KUKA KRL program: f_fraes1.src, f_fraes1.dat

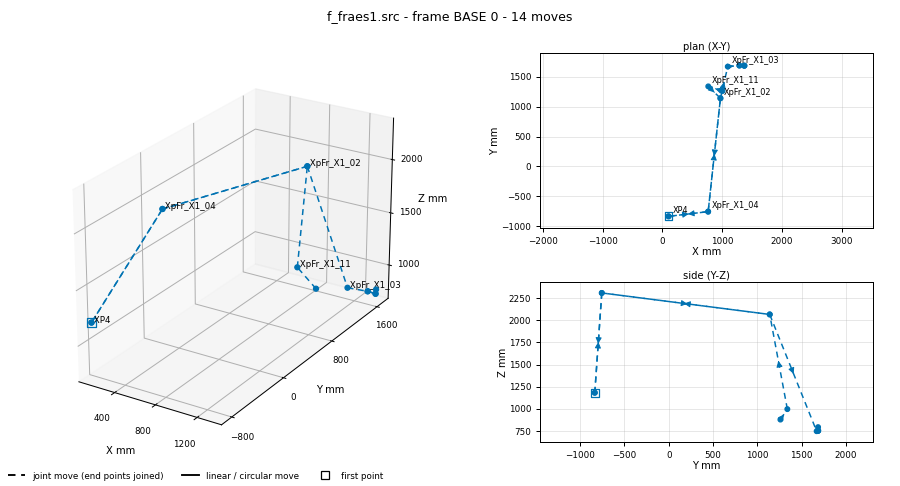
[picture p0: tool path of f_fraes1.src in frame BASE 0, 14 of 15 moves have a stored position in this frame; points joined in program order, loops and branches not executed]
--- f_fraes1.src ---
&ACCESS RVO3
&REL 7
&COMMENT INI Dress X1
&PARAM DISKPATH = KRC:\R1\Program
&PARAM TEMPLATE = C:\KRC\Roboter\Template\vorgabe
&PARAM EDITMASK = *
DEF f_fraes1( )
;FOLD INI
  ;FOLD BASISTECH INI
    GLOBAL INTERRUPT DECL 3 WHEN $STOPMESS==TRUE DO IR_STOPM ( )
    INTERRUPT ON 3
    BAS (#INITMOV,0 )
  ;ENDFOLD (BASISTECH INI)
;FOLD SPOTTECH INI
USERSPOT(#INIT)
;ENDFOLD (SPOTTECH INI)
;FOLD GRIPPERTECH INI
USER_GRP(0,DUMMY,DUMMY,GDEFAULT)
;ENDFOLD (GRIPPERTECH INI)
  ;FOLD USER INI
    ;Make your modifications here

  ;ENDFOLD (USER INI)
;ENDFOLD (INI)

; Caracterização dos meios de produção:
; Versão Atual:
; 08/06/2013 12:00 Name: P13.050-R1 CHANGES: Fresa
; Gun X1 (F2 6640 0018 985)

chk_w1_wechs_ok() ; check X1

;FOLD PTP P4 Vel=100 % PDAT11 Tool[1]:GUN X1 Base[0];%{PE}%R 8.2.20,%MKUKATPBASIS,%CMOVE,%VPTP,%P 1:PTP, 2:P4, 3:, 5:100, 7:PDAT11
$BWDSTART=FALSE
PDAT_ACT=PPDAT11
FDAT_ACT=FP4
BAS(#PTP_PARAMS,100)
PTP XP4
;ENDFOLD

;FOLD PTP pFr_X1_04 CONT Vel=100 % PDAT13 Tool[1]:GUN X1 Base[0];%{PE}%R 8.2.20,%MKUKATPBASIS,%CMOVE,%VPTP,%P 1:PTP, 2:pFr_X1_04, 3:C_DIS, 5:100, 7:PDAT13
$BWDSTART=FALSE
PDAT_ACT=PPDAT13
FDAT_ACT=FpFr_X1_04
BAS(#PTP_PARAMS,100)
PTP XpFr_X1_04 C_DIS
;ENDFOLD
;FOLD PTP pFr_X1_02 CONT Vel=100 % PDAT1 Tool[1]:GUN X1 Base[0];%{PE}%R 8.2.20,%MKUKATPBASIS,%CMOVE,%VPTP,%P 1:PTP, 2:pFr_X1_02, 3:C_DIS, 5:100, 7:PDAT1
$BWDSTART=FALSE
PDAT_ACT=PPDAT1
FDAT_ACT=FpFr_X1_02
BAS(#PTP_PARAMS,100)
PTP XpFr_X1_02 C_DIS
;ENDFOLD
;FOLD PTP pFr_X1_03 CONT Vel=100 % PDAT2 Tool[1]:GUN X1 Base[0];%{PE}%R 8.2.20,%MKUKATPBASIS,%CMOVE,%VPTP,%P 1:PTP, 2:pFr_X1_03, 3:C_DIS, 5:100, 7:PDAT2
$BWDSTART=FALSE
PDAT_ACT=PPDAT2
FDAT_ACT=FpFr_X1_03
BAS(#PTP_PARAMS,100)
PTP XpFr_X1_03 C_DIS
;ENDFOLD
;FOLD PTP pFr_X1_05 CONT Vel=100 % PDAT3 Tool[1]:GUN X1 Base[0];%{PE}%R 8.2.20,%MKUKATPBASIS,%CMOVE,%VPTP,%P 1:PTP, 2:pFr_X1_05, 3:C_DIS, 5:100, 7:PDAT3
$BWDSTART=FALSE
PDAT_ACT=PPDAT3
FDAT_ACT=FpFr_X1_05
BAS(#PTP_PARAMS,100)
PTP XpFr_X1_05 C_DIS
;ENDFOLD
;FOLD LIN pFr_X1_06 Vel=0.25 m/s CPDAT0 Tool[1]:GUN X1 Base[0];%{PE}%R 8.2.20,%MKUKATPBASIS,%CMOVE,%VLIN,%P 1:LIN, 2:pFr_X1_06, 3:, 5:0.25, 7:CPDAT0
$BWDSTART=FALSE
LDAT_ACT=LCPDAT0
FDAT_ACT=FpFr_X1_06
BAS(#CP_PARAMS,0.25)
LIN XpFr_X1_06
;ENDFOLD

;FOLD ; PONTO DE FRESAGEM;%{PE}%R 8.2.20,%MKUKATPBASIS,%CCOMMENT,%VNORMAL,%P 2:PONTO  DE  FRESAGEM
;ENDFOLD
;FOLD TIP.LIN_ Dress5, Spot Gun 4 , RETR open , Tool[1], Base[0], EXT.TCP=FALSE;%{PE}%MKUKATPUSER
FDAT_ACT=FDress5
BAS(#FRAMES)
LIN  XDress5
S_ACT.GUN=4
S_ACT.RETR=#opn
S_READY=FALSE
USERSPOT (#DRESS,S_ACT )
WAIT FOR  S_READY
;ENDFOLD

;FOLD LIN pFr_X1_08 CONT Vel=0.2 m/s CPDAT2 Tool[1]:GUN X1 Base[0];%{PE}%R 8.2.20,%MKUKATPBASIS,%CMOVE,%VLIN,%P 1:LIN, 2:pFr_X1_08, 3:C_DIS C_DIS, 5:0.2, 7:CPDAT2
$BWDSTART=FALSE
LDAT_ACT=LCPDAT2
FDAT_ACT=FpFr_X1_08
BAS(#CP_PARAMS,0.2)
LIN XpFr_X1_08 C_DIS C_DIS
;ENDFOLD
;FOLD LIN pFr_X1_09 CONT Vel=0.35 m/s CPDAT3 Tool[1]:GUN X1 Base[0];%{PE}%R 8.2.20,%MKUKATPBASIS,%CMOVE,%VLIN,%P 1:LIN, 2:pFr_X1_09, 3:C_DIS C_DIS, 5:0.35, 7:CPDAT3
$BWDSTART=FALSE
LDAT_ACT=LCPDAT3
FDAT_ACT=FpFr_X1_09
BAS(#CP_PARAMS,0.35)
LIN XpFr_X1_09 C_DIS C_DIS
;ENDFOLD
;FOLD PTP P3 PDAT10 SPOT Gun=4 RETR OPN PgNo1=254 ACTIVE=1 Tool[1]:GUN X1 Base[1]:Actros;%{PE}%R 8.2.2,%MKUKATPSPOT,%CSPOT,%VPTP,%P 1:PTP, 2:P3, 3:, 5:100, 7:PDAT10, 10:4, 12:#FIRST, 14:#OPN, 16:254, 18:1, 20:0, 22:0, 24:1, 25:NORMAL
$BWDSTART=FALSE
PDAT_ACT=PPDAT10
FDAT_ACT=FP3
BAS(#PTP_PARAMS,PPDAT10.VEL)
S_ACT.GUN=4
S_ACT.PAIR=SDEFAULT.PAIR
S_ACT.RETR=#OPN
S_ACT.CLO_TM=1
S_ACT.PGNO1=254
S_ACT.PGNO2=SDEFAULT.PGNO2
S_ACT.PRESS1=SDEFAULT.PRESS1
S_ACT.PRESS2=SDEFAULT.PRESS2
S_READY=FALSE
PTP XP3
USERSPOT(#SPOT, S_ACT)
WAIT FOR S_READY
;ENDFOLD
;FOLD PTP pFr_X1_10 CONT Vel=100 % PDAT4 Tool[1]:GUN X1 Base[0];%{PE}%R 8.2.20,%MKUKATPBASIS,%CMOVE,%VPTP,%P 1:PTP, 2:pFr_X1_10, 3:C_DIS, 5:100, 7:PDAT4
$BWDSTART=FALSE
PDAT_ACT=PPDAT4
FDAT_ACT=FpFr_X1_10
BAS(#PTP_PARAMS,100)
PTP XpFr_X1_10 C_DIS
;ENDFOLD
;FOLD PTP pFr_X1_11 CONT Vel=100 % PDAT5 Tool[1]:GUN X1 Base[0];%{PE}%R 8.2.20,%MKUKATPBASIS,%CMOVE,%VPTP,%P 1:PTP, 2:pFr_X1_11, 3:C_DIS, 5:100, 7:PDAT5
$BWDSTART=FALSE
PDAT_ACT=PPDAT5
FDAT_ACT=FpFr_X1_11
BAS(#PTP_PARAMS,100)
PTP XpFr_X1_11 C_DIS
;ENDFOLD
;FOLD PTP pFr_X1_12 CONT Vel=100 % PDAT6 Tool[1]:GUN X1 Base[0];%{PE}%R 8.2.20,%MKUKATPBASIS,%CMOVE,%VPTP,%P 1:PTP, 2:pFr_X1_12, 3:C_DIS, 5:100, 7:PDAT6
$BWDSTART=FALSE
PDAT_ACT=PPDAT6
FDAT_ACT=FpFr_X1_12
BAS(#PTP_PARAMS,100)
PTP XpFr_X1_12 C_DIS
;ENDFOLD
;FOLD PTP pFr_X1_07 CONT Vel=100 % PDAT14 Tool[1]:GUN X1 Base[0];%{PE}%R 8.2.20,%MKUKATPBASIS,%CMOVE,%VPTP,%P 1:PTP, 2:pFr_X1_07, 3:C_DIS, 5:100, 7:PDAT14
$BWDSTART=FALSE
PDAT_ACT=PPDAT14
FDAT_ACT=FpFr_X1_07
BAS(#PTP_PARAMS,100)
PTP XpFr_X1_07 C_DIS
;ENDFOLD

;FOLD PTP P5 Vel=100 % PDAT12 Tool[1]:GUN X1 Base[0];%{PE}%R 8.2.20,%MKUKATPBASIS,%CMOVE,%VPTP,%P 1:PTP, 2:P5, 3:, 5:100, 7:PDAT12
$BWDSTART=FALSE
PDAT_ACT=PPDAT12
FDAT_ACT=FP5
BAS(#PTP_PARAMS,100)
PTP XP5
;ENDFOLD

END

--- f_fraes1.dat ---
&ACCESS RVO3
&REL 7
&COMMENT INI Dress X1
&PARAM DISKPATH = KRC:\R1\Program
&PARAM TEMPLATE = C:\KRC\Roboter\Template\vorgabe
&PARAM EDITMASK = *
DEFDAT  f_fraes1
;FOLD EXTERNAL DECLARATIONS;%{PE}%MKUKATPBASIS,%CEXT,%VCOMMON,%P
;FOLD GRIPPERTECH EXT
EXT  H50 (INT  :IN,INT  :IN,INT  :IN,GRP_TYP  :IN )
;ENDFOLD (GRIPPERTECH EXT)
;FOLD SPOTTECH EXT
EXT  USERSPOT (S_COMMAND  :IN,SPOT_TYPE  :IN )
;ENDFOLD (SPOTTECH EXT)
;FOLD BASISTECH EXT;%{PE}%MKUKATPBASIS,%CEXT,%VEXT,%P
EXT  BAS (BAS_COMMAND  :IN,REAL  :IN )
DECL INT SUCCESS
;ENDFOLD (BASISTECH EXT)
;FOLD USER EXT;%{E}%MKUKATPUSER,%CEXT,%VEXT,%P
;Make your modifications here

;ENDFOLD (USER EXT)
;ENDFOLD (EXTERNAL DECLARATIONS)
DECL BASIS_SUGG_T LAST_BASIS={POINT1[] "P5                      ",POINT2[] "P5                      ",CP_PARAMS[] "CPDAT3                  ",PTP_PARAMS[] "PDAT14                  ",CONT[] "                        ",CP_VEL[] "0.35                    ",PTP_VEL[] "100                     ",SYNC_PARAMS[] "SYNCDAT                 ",SPL_NAME[] "S0                      "}
DECL PDAT PPDAT1={VEL 100.0,ACC 100.0,APO_DIST 100.0,APO_MODE #CDIS}
DECL E6POS XpFr_X1_02={X 969.039673,Y 1139.73096,Z 2066.15308,A 44.3954697,B 54.7452507,C 92.8609467,S 2,T 3,E1 199.989594,E2 0.0,E3 0.0,E4 0.0,E5 0.0,E6 0.0}
DECL FDAT FpFr_X1_02={TOOL_NO 1,BASE_NO 0,IPO_FRAME #BASE,POINT2[] " ",TQ_STATE FALSE}
DECL PDAT PPDAT2={VEL 100.0,ACC 100.0,APO_DIST 100.0,APO_MODE #CDIS}
DECL E6POS XpFr_X1_03={X 1091.45203,Y 1668.95398,Z 749.063171,A 0.738173604,B 22.6249809,C -0.268216789,S 2,T 35,E1 -532.459717,E2 0.0,E3 0.0,E4 0.0,E5 0.0,E6 0.0}
DECL FDAT FpFr_X1_03={TOOL_NO 1,BASE_NO 0,IPO_FRAME #BASE,POINT2[] " ",TQ_STATE FALSE}
DECL PDAT PPDAT3={VEL 100.0,ACC 100.0,APO_DIST 100.0,APO_MODE #CDIS}
DECL E6POS XpFr_X1_05={X 1286.05005,Y 1686.81702,Z 755.587097,A 0.624875784,B 1.75245798,C 1.14266706,S 2,T 35,E1 -532.457886,E2 0.0,E3 0.0,E4 0.0,E5 0.0,E6 0.0}
DECL FDAT FpFr_X1_05={TOOL_NO 1,BASE_NO 0,IPO_FRAME #BASE,POINT2[] " ",TQ_STATE FALSE}
DECL LDAT LCPDAT0={VEL 2.0,ACC 100.0,APO_DIST 100.0,APO_FAC 50.0,AXIS_VEL 100.0,AXIS_ACC 100.0,ORI_TYP #VAR,CIRC_TYP #BASE,JERK_FAC 50.0,GEAR_JERK 50.0,EXAX_IGN 0}
DECL E6POS XpFr_X1_06={X 1368.19702,Y 1682.95203,Z 753.130981,A 0.624874711,B 1.75245702,C 1.14266706,S 2,T 35,E1 -532.457581,E2 0.0,E3 0.0,E4 0.0,E5 0.0,E6 0.0}
DECL FDAT FpFr_X1_06={TOOL_NO 1,BASE_NO 0,IPO_FRAME #BASE,POINT2[] " ",TQ_STATE FALSE}
DECL SPOT_SUGG_T LAST_SPOT={GUN[] "4                       ",RETR_CMD[] "#OPN                    ",CHOISE[] "#FIRST                  ",CLO_TM[] "1                       ",PGNO1[] "1                       ",PRESS1[] "0                       ",PGNO2[] "1                       ",PRESS2[] "0                       ",SPOT_PARAMS[] "NORMAL                  "}
DECL LDAT LCPDAT2={VEL 2.0,ACC 100.0,APO_DIST 100.0,APO_FAC 50.0,AXIS_VEL 100.0,AXIS_ACC 100.0,ORI_TYP #VAR,CIRC_TYP #BASE,JERK_FAC 50.0,GEAR_JERK 50.0,EXAX_IGN 0}
DECL E6POS XpFr_X1_08={X 1366.25,Y 1684.50903,Z 753.133484,A 0.625003517,B 1.75241804,C 1.14276195,S 2,T 35,E1 -532.457825,E2 0.0,E3 0.0,E4 0.0,E5 0.0,E6 0.0}
DECL FDAT FpFr_X1_08={TOOL_NO 1,BASE_NO 0,IPO_FRAME #BASE,POINT2[] " ",TQ_STATE FALSE}
DECL LDAT LCPDAT3={VEL 2.0,ACC 100.0,APO_DIST 100.0,APO_FAC 50.0,AXIS_VEL 100.0,AXIS_ACC 100.0,ORI_TYP #VAR,CIRC_TYP #BASE,JERK_FAC 50.0,GEAR_JERK 50.0,EXAX_IGN 0}
DECL E6POS XpFr_X1_09={X 1286.05005,Y 1686.81702,Z 755.587219,A 0.624872983,B 1.75245202,C 1.14266598,S 2,T 35,E1 -532.457886,E2 0.0,E3 0.0,E4 0.0,E5 0.0,E6 0.0}
DECL FDAT FpFr_X1_09={TOOL_NO 1,BASE_NO 0,IPO_FRAME #BASE,POINT2[] " ",TQ_STATE FALSE}
DECL PDAT PPDAT4={VEL 100.0,ACC 100.0,APO_DIST 100.0,APO_MODE #CDIS}
DECL E6POS XpFr_X1_10={X 1003.46301,Y 1260.20398,Z 880.076172,A 5.04273415,B 32.9262886,C 2.90043402,S 2,T 35,E1 -382.985596,E2 0.0,E3 0.0,E4 0.0,E5 0.0,E6 0.0}
DECL FDAT FpFr_X1_10={TOOL_NO 1,BASE_NO 0,IPO_FRAME #BASE,POINT2[] " ",TQ_STATE FALSE}
DECL PDAT PPDAT5={VEL 100.0,ACC 100.0,APO_DIST 100.0,APO_MODE #CDIS}
DECL E6POS XpFr_X1_11={X 765.945618,Y 1338.37,Z 998.083374,A 14.9633598,B 64.6672592,C 12.7722797,S 2,T 3,E1 -223.039795,E2 0.0,E3 0.0,E4 0.0,E5 0.0,E6 0.0}
DECL FDAT FpFr_X1_11={TOOL_NO 1,BASE_NO 0,IPO_FRAME #BASE,POINT2[] " ",TQ_STATE FALSE}
DECL PDAT PPDAT6={VEL 100.0,ACC 100.0,APO_DIST 100.0,APO_MODE #CDIS}
DECL E6POS XpFr_X1_12={X 969.039673,Y 1139.73096,Z 2066.15308,A 44.3954697,B 54.7452507,C 92.8609467,S 2,T 3,E1 199.989594,E2 0.0,E3 0.0,E4 0.0,E5 0.0,E6 0.0}
DECL FDAT FpFr_X1_12={TOOL_NO 1,BASE_NO 0,IPO_FRAME #BASE,POINT2[] " ",TQ_STATE FALSE}
DECL FDAT FDress5={TOOL_NO 1,BASE_NO 0,IPO_FRAME #BASE}
DECL E6POS XDress5={X 1370.49097,Y 1685.20703,Z 794.879211,A 0.670950472,B 1.68890405,C 0.515060484,S 2,T 35,E1 -532.459106,E2 0.0,E3 0.0,E4 0.0,E5 0.0,E6 0.0}
DECL E6POS XP3={X 9762.19434,Y -3811.4519,Z -756.436829,A -89.2618332,B 22.6249809,C -0.268216789,S 2,T 35,E1 -532.459717,E2 0.0,E3 0.0,E4 0.0,E5 0.0,E6 0.0}
DECL FDAT FP3={TOOL_NO 1,BASE_NO 1,IPO_FRAME #BASE,POINT2[] " ",TQ_STATE FALSE}
DECL PDAT PPDAT10={VEL 100.0,ACC 100.0,APO_DIST 100.0,APO_MODE #CDIS}
DECL E6POS XP4={X 101.904198,Y -833.887207,Z 1182.97998,A -87.0955505,B 79.0952911,C 80.3321075,S 2,T 2,E1 213.625793,E2 0.0,E3 0.0,E4 0.0,E5 0.0,E6 0.0}
DECL FDAT FP4={TOOL_NO 1,BASE_NO 0,IPO_FRAME #BASE,POINT2[] " ",TQ_STATE FALSE}
DECL PDAT PPDAT11={VEL 100.0,ACC 100.0,APO_DIST 100.0,APO_MODE #CDIS}
DECL E6POS XP5={X 101.904198,Y -833.887207,Z 1182.97998,A -87.0955505,B 79.0952911,C 80.3321075,S 2,T 2,E1 213.625793,E2 0.0,E3 0.0,E4 0.0,E5 0.0,E6 0.0}
DECL FDAT FP5={TOOL_NO 1,BASE_NO 0,IPO_FRAME #BASE,POINT2[] " ",TQ_STATE FALSE}
DECL PDAT PPDAT12={VEL 100.0,ACC 100.0,APO_DIST 100.0,APO_MODE #CDIS}
DECL PDAT PPDAT13={VEL 100.0,ACC 100.0,APO_DIST 100.0,APO_MODE #CDIS}
DECL E6POS XpFr_X1_04={X 763.830505,Y -754.804016,Z 2308.69702,A -54.2272797,B 44.6665993,C 55.8185196,S 2,T 3,E1 207.1996,E2 0.0,E3 0.0,E4 0.0,E5 0.0,E6 0.0}
DECL FDAT FpFr_X1_04={TOOL_NO 1,BASE_NO 0,IPO_FRAME #BASE,POINT2[] " ",TQ_STATE FALSE}
DECL PDAT PPDAT14={VEL 100.0,ACC 100.0,APO_DIST 100.0,APO_MODE #CDIS}
DECL E6POS XpFr_X1_07={X 763.830505,Y -754.804016,Z 2308.69702,A -54.2272797,B 44.6665993,C 55.8185196,S 2,T 3,E1 207.1996,E2 0.0,E3 0.0,E4 0.0,E5 0.0,E6 0.0}
DECL FDAT FpFr_X1_07={TOOL_NO 1,BASE_NO 0,IPO_FRAME #BASE,POINT2[] " ",TQ_STATE FALSE}
ENDDAT
